// TIA Portal project "Tank_1" (V20)

(* hardware
DEVICE "S7-1500/ET200MP-Station_1"  S7-1500 station
   slot 0: "Profilschiene_0"  Rack  6ES7 590-1***0-0AA0
   slot 1: "PLC_1"  CPU 1513-1 PN  6ES7 513-1AM03-0AB0  V4.0
      slot 3: "CPU-Display_1"  6ES7591-1AA00-0AA0
      slot 32768: "PROFINET-Schnittstelle_1"  X1
         slot 32769: "Port_1"  X1 P1
         slot 32770: "Port_2"  X1 P2
      slot 34817: "Virtual CP interface port_1"  Virtual CP interface port  Virtual CP interface port FW V4.0
   slot 2: "DI 16x24VDC BA_1"  DI 16x24VDC BA  6ES7 521-1BH10-0AA0  V1.1
   slot 3: "DQ 16x24VDC/0.5A ST_1"  DQ 16x24VDC/0.5A ST  6ES7 522-1BH00-0AB0  V2.0
   slot 4: "AI 8xU/I/R/RTD BA_1"  AI 8xU/I/R/RTD BA  6ES7 531-7QF00-0AB0  V1.0
   slot 5: "AQ 8xU/I HS_1"  AQ 8xU/I HS  6ES7 532-5HF00-0AB0  V2.2
*)

// ===== PLC "PLC_1"  CPU 1513-1 PN =====

VAR_GLOBAL   // PLC tag table "Standard-Variablentabelle"
   "PlcLabConnectIn01" AT %ID32760 : DWord;
   "PlcLabConnectIn02" AT %ID32764 : DWord;
   "PlcLabConnectOut01" AT %QD32760 : DWord;
   "PlcLabConnectOut02" AT %QD32764 : DWord;
   "Durchmesser_Tank" AT %MD40 : Real;
   "Hoehe_Tank" AT %MD44 : Real;
   "Aktuelle_Fuellhoehe" AT %MD52 : Real;
   "Max_Fuellstand" AT %MD48 : Real;
   "Aktueller_Fuellstand" AT %MD56 : Real;
   "Fuellstand_Prozent" AT %MD60 : Real;
END_VAR

DATA_BLOCK "DB_1"   // DB1
{ S7_Optimized_Access := 'TRUE' }
VERSION : 0.1
   VAR
      Tanks : Struct
         Tank_1 : Struct
            Durchmesser : Real := 3.0;
            Hoehe : Real := 4.0;
            Max_Fuellstand : Real;
            Akt_Fuellhoehe : Real := 2.5;
            Akt_Fuellstand : Real;
            Fuellstand_Prozent : Real;
         END_STRUCT;
         Tank_2 : Struct
            Durchmesser : Real := 4.0;
            Hoehe : Real := 4.0;
            Max_Fuellstand : Real;
            Akt_Fuellhoehe : Real := 2.5;
            Akt_Fuellstand : Real;
            Fuellstand_Prozent : Real;
         END_STRUCT;
         Tank_3 : Struct
            Durchmesser : Real := 2.5;
            Hoehe : Real := 4.0;
            Max_Fuellstand : Real;
            Akt_Fuellhoehe : Real := 2.5;
            Akt_Fuellstand : Real;
            Fuellstand_Prozent : Real;
         END_STRUCT;
      END_STRUCT;
   END_VAR
BEGIN
END_DATA_BLOCK

FUNCTION "Tankberechnung" : Void   // FC1, FBD
{ S7_Optimized_Access := 'TRUE' }
VERSION : 0.1
   VAR_INPUT
      Durchmesser : Real;
      Hoehe : Real;
      Fuellhoehe : Real;
   END_VAR
   VAR_OUTPUT
      Fuellstand_Prozent : Real;
   END_VAR
   VAR_IN_OUT
      Maximum : Real;
      Fuellstand : Real;
   END_VAR
   VAR CONSTANT
      PI : Real := 3.14153;
      Teiler_d : Real := 2.0;   // Um den Durchmesser in den Radius zu wandeln.
      Einheit_l : Real := 1000.0;   // Um von Kubikmeter in Liter umzurechnen
   END_VAR
BEGIN

REGION Network 1
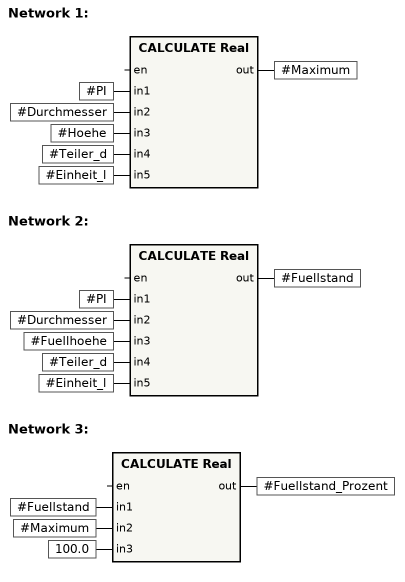
   #Maximum := #PI * ((#Durchmesser / #Teiler_d) * (#Durchmesser / #Teiler_d)) * #Hoehe * #Einheit_l;
END_REGION

REGION Network 2
   #Fuellstand := #PI * ((#Durchmesser / #Teiler_d) * (#Durchmesser / #Teiler_d)) * #Fuellhoehe * #Einheit_l;
END_REGION

REGION Network 3
   #Fuellstand_Prozent := (#Fuellstand / #Maximum) * 100.0;
END_REGION
END_FUNCTION

ORGANIZATION_BLOCK "Main"   // OB1, FBD, ProgramCycle
TITLE = "Main Program Sweep (Cycle)"
{ S7_Optimized_Access := 'TRUE' }
VERSION : 0.1
   VAR_INPUT
      Initial_Call : Bool;   // Initial call of this OB
      Remanence : Bool;   // =True, if remanent data are available
   END_VAR
BEGIN

REGION Network 1
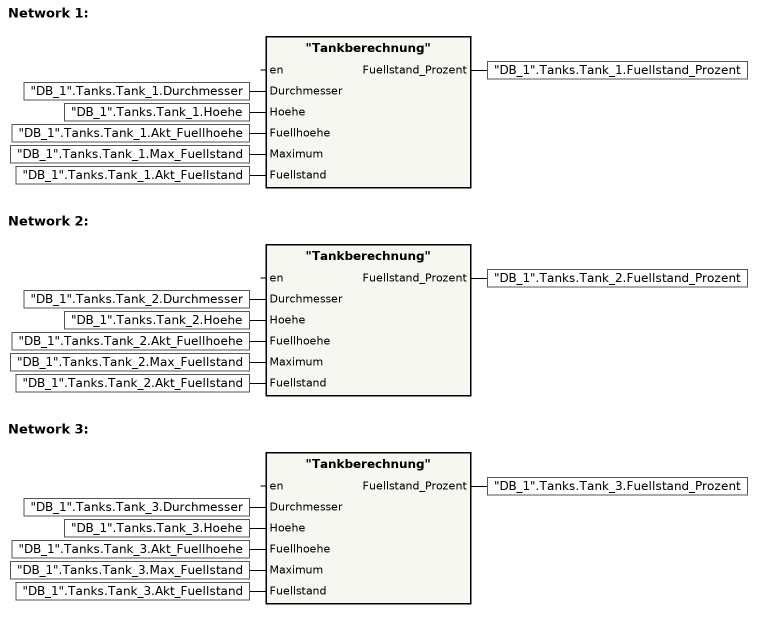
   "Tankberechnung"(Durchmesser := "DB_1".Tanks.Tank_1.Durchmesser,
                    Hoehe := "DB_1".Tanks.Tank_1.Hoehe,
                    Fuellhoehe := "DB_1".Tanks.Tank_1.Akt_Fuellhoehe,
                    Maximum := "DB_1".Tanks.Tank_1.Max_Fuellstand,
                    Fuellstand := "DB_1".Tanks.Tank_1.Akt_Fuellstand,
                    Fuellstand_Prozent => "DB_1".Tanks.Tank_1.Fuellstand_Prozent);
END_REGION

REGION Network 2
   "Tankberechnung"(Durchmesser := "DB_1".Tanks.Tank_2.Durchmesser,
                    Hoehe := "DB_1".Tanks.Tank_2.Hoehe,
                    Fuellhoehe := "DB_1".Tanks.Tank_2.Akt_Fuellhoehe,
                    Maximum := "DB_1".Tanks.Tank_2.Max_Fuellstand,
                    Fuellstand := "DB_1".Tanks.Tank_2.Akt_Fuellstand,
                    Fuellstand_Prozent => "DB_1".Tanks.Tank_2.Fuellstand_Prozent);
END_REGION

REGION Network 3
   "Tankberechnung"(Durchmesser := "DB_1".Tanks.Tank_3.Durchmesser,
                    Hoehe := "DB_1".Tanks.Tank_3.Hoehe,
                    Fuellhoehe := "DB_1".Tanks.Tank_3.Akt_Fuellhoehe,
                    Maximum := "DB_1".Tanks.Tank_3.Max_Fuellstand,
                    Fuellstand := "DB_1".Tanks.Tank_3.Akt_Fuellstand,
                    Fuellstand_Prozent => "DB_1".Tanks.Tank_3.Fuellstand_Prozent);
END_REGION
END_ORGANIZATION_BLOCK